KUKA KRL program: GlobalPosn.sub, GlobalPosn.dat

--- GlobalPosn.sub ---
&ACCESS RVO1
&REL 1
&PARAM EDITMASK = *
&PARAM TEMPLATE = C:\KRC\Roboter\Template\submit
DEF  GlobalPosn ( )
; **************************************
; * Package:     TeslaCore             *
; * Release      V4.0.0                *
; * File:        GlobalPosn.sub        *
; * Date:        07.2016               *
; * GUI Version: > = V8.3              *
; **************************************
;FOLD Details
;FOLD Declaration
DECL BOOL bPosEvalResult
;ENDFOLD (Declaration)
LOOP
;FOLD Implementation
;FOLD Position GP1
IF (xGP_Ctrl[1].PosnEnabled==TRUE) THEN
	bPosEvalResult = CheckAxisPos(XGlobal1,xGP_Ctrl[1])
	SetPosOut(bPosEvalResult,xGP_Ctrl[1])
ELSE
   SetPosOut(FALSE,xGP_Ctrl[1])
ENDIF
;ENDFOLD (Position GP1)
;FOLD Position GP2
IF (xGP_Ctrl[2].PosnEnabled==TRUE) THEN
	bPosEvalResult = CheckAxisPos(XGlobal2,xGP_Ctrl[2])
	SetPosOut(bPosEvalResult,xGP_Ctrl[2])
ELSE
   SetPosOut(FALSE,xGP_Ctrl[2])
ENDIF
;ENDFOLD (Position GP2)
;FOLD Position GP3
IF (xGP_Ctrl[3].PosnEnabled==TRUE) THEN
	bPosEvalResult = CheckAxisPos(XGlobal3,xGP_Ctrl[3])
	SetPosOut(bPosEvalResult,xGP_Ctrl[3])
ELSE
   SetPosOut(FALSE,xGP_Ctrl[3])
ENDIF
;ENDFOLD (Position GP3)
;FOLD Position GP4
IF (xGP_Ctrl[4].PosnEnabled==TRUE) THEN
	bPosEvalResult = CheckAxisPos(XGlobal4,xGP_Ctrl[4])
	SetPosOut(bPosEvalResult,xGP_Ctrl[4])
ELSE
   SetPosOut(FALSE,xGP_Ctrl[4])
ENDIF
;ENDFOLD (Position GP4)
;FOLD Position GP5
IF (xGP_Ctrl[5].PosnEnabled==TRUE) THEN
	bPosEvalResult = CheckAxisPos(XGlobal5,xGP_Ctrl[5])
	SetPosOut(bPosEvalResult,xGP_Ctrl[5])
ELSE
   SetPosOut(FALSE,xGP_Ctrl[5])
ENDIF
;ENDFOLD (Position GP5)
;FOLD Position GP6
IF (xGP_Ctrl[6].PosnEnabled==TRUE) THEN
	bPosEvalResult = CheckAxisPos(XGlobal6,xGP_Ctrl[6])
	SetPosOut(bPosEvalResult,xGP_Ctrl[6])
ELSE
   SetPosOut(FALSE,xGP_Ctrl[6])
ENDIF
;ENDFOLD (Position GP6)
;FOLD Position GP7
IF (xGP_Ctrl[7].PosnEnabled==TRUE) THEN
	bPosEvalResult = CheckAxisPos(XGlobal7,xGP_Ctrl[7])
	SetPosOut(bPosEvalResult,xGP_Ctrl[7])
ELSE
   SetPosOut(FALSE,xGP_Ctrl[7])
ENDIF
;ENDFOLD (Position GP7)
;FOLD Position GP8
IF (xGP_Ctrl[8].PosnEnabled==TRUE) THEN
	bPosEvalResult = CheckAxisPos(XGlobal8,xGP_Ctrl[8])
	SetPosOut(bPosEvalResult,xGP_Ctrl[8])
ELSE
   SetPosOut(FALSE,xGP_Ctrl[8])
ENDIF
;ENDFOLD (Position GP8)
;FOLD Position GP9
IF (xGP_Ctrl[9].PosnEnabled==TRUE) THEN
	bPosEvalResult = CheckAxisPos(XGlobal9,xGP_Ctrl[9])
	SetPosOut(bPosEvalResult,xGP_Ctrl[9])
ELSE
   SetPosOut(FALSE,xGP_Ctrl[9])
ENDIF
;ENDFOLD (Position GP9)
;FOLD Position GP10
IF (xGP_Ctrl[10].PosnEnabled==TRUE) THEN
	bPosEvalResult = CheckAxisPos(XGlobal10,xGP_Ctrl[10])
	SetPosOut(bPosEvalResult,xGP_Ctrl[10])
ELSE
   SetPosOut(FALSE,xGP_Ctrl[10])
ENDIF
;ENDFOLD (Position GP10)
;ENDFOLD (Implementation)
ENDLOOP
;ENDFOLD (Details)
END ; (GlobalPosn)

DEFFCT BOOL CheckAxisPos (pPosition: IN, pPosCtrl: IN )
;FOLD Details
;FOLD Declaration
E6Axis pPosition
DECL PosnCtrl_Typ pPosCtrl
BOOL bResult
REAL Angle1, Angle2, Angle3, Angle4, Angle5, Angle6, Angle7, Angle8, Angle9, Angle10, Angle11, Angle12
;ENDFOLD (Declaration)
;FOLD Implementation
IF ((VARSTATE("pPosition") == #INITIALIZED) AND (VARSTATE("pPosCtrl") == #INITIALIZED))THEN
	Angle1 =  ABS(pPosition.A1 - $AXIS_ACT.A1)
	IF (Angle1>pPosCtrl.A1_Tol) THEN
		RETURN(FALSE)
	ENDIF
	Angle2 =  ABS(pPosition.A2 - $AXIS_ACT.A2)
	IF (Angle2>pPosCtrl.A2_Tol) THEN
		RETURN(FALSE)
	ENDIF
	Angle3 =  ABS(pPosition.A3 - $AXIS_ACT.A3)
	IF (Angle3>pPosCtrl.A3_Tol) THEN
		RETURN(FALSE)
	ENDIF
	Angle4 =  ABS(pPosition.A4 - $AXIS_ACT.A4)
	IF (Angle4>pPosCtrl.A4_Tol) THEN
		RETURN(FALSE)
	ENDIF
	Angle5 =  ABS(pPosition.A5 - $AXIS_ACT.A5)
	IF (Angle5>pPosCtrl.A5_Tol) THEN
		RETURN(FALSE)
	ENDIF
	Angle6 =  ABS(pPosition.A6 - $AXIS_ACT.A6)
	IF (Angle6>pPosCtrl.A6_Tol) THEN
		RETURN(FALSE)
	ENDIF
	Angle7 =  ABS(pPosition.E1 - $AXIS_ACT.E1)
	IF (Angle7>pPosCtrl.E1_Tol) THEN
		RETURN(FALSE)
	ENDIF
	Angle8 =  ABS(pPosition.E2 - $AXIS_ACT.E2)
	IF (Angle8>pPosCtrl.E2_Tol) THEN
		RETURN(FALSE)
	ENDIF
	Angle9 =  ABS(pPosition.E3 - $AXIS_ACT.E3)
	IF (Angle9>pPosCtrl.E3_Tol) THEN
		RETURN(FALSE)
	ENDIF
	Angle10 =  ABS(pPosition.E4 - $AXIS_ACT.E4)
	IF (Angle10>pPosCtrl.E4_Tol) THEN
		RETURN(FALSE)
	ENDIF
	Angle11 =  ABS(pPosition.E5 - $AXIS_ACT.E5)
	IF (Angle11>pPosCtrl.E5_Tol) THEN
		RETURN(FALSE)
	ENDIF
	Angle12 =  ABS(pPosition.E6 - $AXIS_ACT.E6)
	IF (Angle12>pPosCtrl.E6_Tol) THEN
		RETURN(FALSE)
	ENDIF
	RETURN (TRUE)
ELSE
	RETURN (FALSE)
ENDIF
;ENDFOLD (Implementation)
;ENDFOLD (Details)
ENDFCT ; (CheckAxisPos)

DEF SetPosOut(bState :IN, pPosCtrl :IN)
;FOLD Details
;FOLD Declaration
BOOL bState
DECL PosnCtrl_Typ pPosCtrl
;ENDFOLD (Declaration)
;FOLD Implementation
IF ((VARSTATE("bState") == #INITIALIZED) AND (VARSTATE("pPosCtrl") == #INITIALIZED))THEN
	IF (pPosCtrl.OutputCtrl > 0) THEN
		IF (pPosCtrl.AtPosn == TRUE) THEN
			$OUT[pPosCtrl.OutputCtrl]=bState
		ELSE
			$OUT[pPosCtrl.OutputCtrl]=NOT(bState)
		ENDIF
	ENDIF
ENDIF
;ENDFOLD (Implementation)
;ENDFOLD (Details)
END ; (SetPosOut)

--- GlobalPosn.dat ---
&ACCESS RVO1
&REL 1
&PARAM EDITMASK = *
&PARAM TEMPLATE = C:\KRC\Roboter\Template\submit
DEFDAT GlobalPosn PUBLIC
; **************************************
; * Package:     TeslaCore             *
; * Release      V4.0.0                *
; * File:        GlobalPosn.dat        *
; * Date:        07.2016               *
; * GUI Version: > = V8.3              *
; **************************************

;FOLD Control Information
DECL GLOBAL INT nMaxGlobalPosn=10 ; Maximum # of global positions
GLOBAL STRUC PosnCtrl_Typ CHAR Comment[24], BOOL PosnEnabled,AtPosn, INT OutputCtrl, REAL A1_Tol, A2_Tol, A3_Tol, A4_Tol, A5_Tol, A6_Tol, E1_Tol, E2_Tol, E3_Tol, E4_Tol, E5_Tol, E6_Tol
DECL GLOBAL PosnCtrl_Typ xGP_Ctrl[10]
xGP_Ctrl[1]={Comment[]" ", PosnEnabled FALSE, AtPosn FALSE, OutputCtrl 0, A1_Tol 2.0, A2_Tol 2.0, A3_Tol 2.0, A4_Tol 2.0, A5_Tol 2.0, A6_Tol 2.0, E1_Tol 2.0, E2_Tol 2.0, E3_Tol 2.0, E4_Tol 2.0, E5_Tol 2.0, E6_Tol 2.0}
xGP_Ctrl[2]={Comment[]" ", PosnEnabled FALSE, AtPosn FALSE,OutputCtrl 0, A1_Tol 2.0, A2_Tol 2.0, A3_Tol 2.0, A4_Tol 2.0, A5_Tol 2.0, A6_Tol 2.0, E1_Tol 2.0, E2_Tol 2.0, E3_Tol 2.0, E4_Tol 2.0, E5_Tol 2.0, E6_Tol 2.0}
xGP_Ctrl[3]={Comment[]" ", PosnEnabled FALSE, AtPosn FALSE,OutputCtrl 0, A1_Tol 2.0, A2_Tol 2.0, A3_Tol 2.0, A4_Tol 2.0, A5_Tol 2.0, A6_Tol 2.0, E1_Tol 2.0, E2_Tol 2.0, E3_Tol 2.0, E4_Tol 2.0, E5_Tol 2.0, E6_Tol 2.0}
xGP_Ctrl[4]={Comment[]" ", PosnEnabled FALSE, AtPosn FALSE,OutputCtrl 0, A1_Tol 2.0, A2_Tol 2.0, A3_Tol 2.0, A4_Tol 2.0, A5_Tol 2.0, A6_Tol 2.0, E1_Tol 2.0, E2_Tol 2.0, E3_Tol 2.0, E4_Tol 2.0, E5_Tol 2.0, E6_Tol 2.0}
xGP_Ctrl[5]={Comment[]" ", PosnEnabled FALSE, AtPosn FALSE,OutputCtrl 0, A1_Tol 2.0, A2_Tol 2.0, A3_Tol 2.0, A4_Tol 2.0, A5_Tol 2.0, A6_Tol 2.0, E1_Tol 2.0, E2_Tol 2.0, E3_Tol 2.0, E4_Tol 2.0, E5_Tol 2.0, E6_Tol 2.0}
xGP_Ctrl[6]={Comment[]" ", PosnEnabled FALSE, AtPosn FALSE,OutputCtrl 0, A1_Tol 2.0, A2_Tol 2.0, A3_Tol 2.0, A4_Tol 2.0, A5_Tol 2.0, A6_Tol 2.0, E1_Tol 2.0, E2_Tol 2.0, E3_Tol 2.0, E4_Tol 2.0, E5_Tol 2.0, E6_Tol 2.0}
xGP_Ctrl[7]={Comment[]" ", PosnEnabled FALSE, AtPosn FALSE,OutputCtrl 0, A1_Tol 2.0, A2_Tol 2.0, A3_Tol 2.0, A4_Tol 2.0, A5_Tol 2.0, A6_Tol 2.0, E1_Tol 2.0, E2_Tol 2.0, E3_Tol 2.0, E4_Tol 2.0, E5_Tol 2.0, E6_Tol 2.0}
xGP_Ctrl[8]={Comment[]" ", PosnEnabled FALSE, AtPosn FALSE,OutputCtrl 0, A1_Tol 2.0, A2_Tol 2.0, A3_Tol 2.0, A4_Tol 2.0, A5_Tol 2.0, A6_Tol 2.0, E1_Tol 2.0, E2_Tol 2.0, E3_Tol 2.0, E4_Tol 2.0, E5_Tol 2.0, E6_Tol 2.0}
xGP_Ctrl[9]={Comment[]" ", PosnEnabled FALSE, AtPosn FALSE,OutputCtrl 0, A1_Tol 2.0, A2_Tol 2.0, A3_Tol 2.0, A4_Tol 2.0, A5_Tol 2.0, A6_Tol 2.0, E1_Tol 2.0, E2_Tol 2.0, E3_Tol 2.0, E4_Tol 2.0, E5_Tol 2.0, E6_Tol 2.0}
xGP_Ctrl[10]={Comment[]" ", PosnEnabled FALSE, AtPosn FALSE,OutputCtrl 0, A1_Tol 2.0, A2_Tol 2.0, A3_Tol 2.0, A4_Tol 2.0, A5_Tol 2.0, A6_Tol 2.0, E1_Tol 2.0, E2_Tol 2.0, E3_Tol 2.0, E4_Tol 2.0, E5_Tol 2.0, E6_Tol 2.0}
;ENDFOLD (Control Information)
;FOLD Positional Information
DECL GLOBAL E6AXIS XGlobal1={A1 0.0,A2 -90.0,A3 90.0,A4 0.0,A5 0.0,A6 0.0,E1 0.0,E2 0.0,E3 0.0,E4 0.0,E5 0.0,E6 0.0}
DECL GLOBAL FDAT FGlobal1={TOOL_NO 1,BASE_NO 0,IPO_FRAME #BASE,POINT2[] " ",TQ_STATE FALSE}
DECL GLOBAL PDAT PGlobal1={VEL 100.000,ACC 100.000,APO_DIST 100.000,GEAR_JERK 50.0000}
DECL GLOBAL LDAT LCGlobal1={VEL 2.00000,ACC 100.000,APO_DIST 100.000,APO_FAC 50.0000,AXIS_VEL 100.000,AXIS_ACC 100.000,ORI_TYP #VAR,CIRC_TYP #BASE,JERK_FAC 50.0000,GEAR_JERK 50.0000,EXAX_IGN 0}

DECL GLOBAL E6AXIS XGlobal2={A1 0.0,A2 -90.0,A3 90.0,A4 0.0,A5 0.0,A6 0.0,E1 0.0,E2 0.0,E3 0.0,E4 0.0,E5 0.0,E6 0.0}
DECL GLOBAL FDAT FGlobal2={TOOL_NO 1,BASE_NO 0,IPO_FRAME #BASE,POINT2[] " ",TQ_STATE FALSE}
DECL GLOBAL PDAT PGlobal2={VEL 100.000,ACC 100.000,APO_DIST 100.000,GEAR_JERK 50.0000}
DECL GLOBAL LDAT LCGlobal2={VEL 2.00000,ACC 100.000,APO_DIST 100.000,APO_FAC 50.0000,AXIS_VEL 100.000,AXIS_ACC 100.000,ORI_TYP #VAR,CIRC_TYP #BASE,JERK_FAC 50.0000,GEAR_JERK 50.0000,EXAX_IGN 0}

DECL GLOBAL E6AXIS XGlobal3={A1 0.0,A2 -90.0,A3 90.0,A4 0.0,A5 0.0,A6 0.0,E1 0.0,E2 0.0,E3 0.0,E4 0.0,E5 0.0,E6 0.0}
DECL GLOBAL FDAT FGlobal3={TOOL_NO 1,BASE_NO 0,IPO_FRAME #BASE,POINT2[] " ",TQ_STATE FALSE}
DECL GLOBAL PDAT PGlobal3={VEL 100.000,ACC 100.000,APO_DIST 100.000,GEAR_JERK 50.0000}
DECL GLOBAL LDAT LCGlobal3={VEL 2.00000,ACC 100.000,APO_DIST 100.000,APO_FAC 50.0000,AXIS_VEL 100.000,AXIS_ACC 100.000,ORI_TYP #VAR,CIRC_TYP #BASE,JERK_FAC 50.0000,GEAR_JERK 50.0000,EXAX_IGN 0}

DECL GLOBAL E6AXIS XGlobal4={A1 0.0,A2 -90.0,A3 90.0,A4 0.0,A5 0.0,A6 0.0,E1 0.0,E2 0.0,E3 0.0,E4 0.0,E5 0.0,E6 0.0}
DECL GLOBAL FDAT FGlobal4={TOOL_NO 1,BASE_NO 0,IPO_FRAME #BASE,POINT2[] " ",TQ_STATE FALSE}
DECL GLOBAL PDAT PGlobal4={VEL 100.000,ACC 100.000,APO_DIST 100.000,GEAR_JERK 50.0000}
DECL GLOBAL LDAT LCGlobal4={VEL 2.00000,ACC 100.000,APO_DIST 100.000,APO_FAC 50.0000,AXIS_VEL 100.000,AXIS_ACC 100.000,ORI_TYP #VAR,CIRC_TYP #BASE,JERK_FAC 50.0000,GEAR_JERK 50.0000,EXAX_IGN 0}

DECL GLOBAL E6AXIS XGlobal5={A1 0.0,A2 -90.0,A3 90.0,A4 0.0,A5 0.0,A6 0.0,E1 0.0,E2 0.0,E3 0.0,E4 0.0,E5 0.0,E6 0.0}
DECL GLOBAL FDAT FGlobal5={TOOL_NO 1,BASE_NO 0,IPO_FRAME #BASE,POINT2[] " ",TQ_STATE FALSE}
DECL GLOBAL PDAT PGlobal5={VEL 100.000,ACC 100.000,APO_DIST 100.000,GEAR_JERK 50.0000}
DECL GLOBAL LDAT LCGlobal5={VEL 2.00000,ACC 100.000,APO_DIST 100.000,APO_FAC 50.0000,AXIS_VEL 100.000,AXIS_ACC 100.000,ORI_TYP #VAR,CIRC_TYP #BASE,JERK_FAC 50.0000,GEAR_JERK 50.0000,EXAX_IGN 0}

DECL GLOBAL E6AXIS XGlobal6={A1 0.0,A2 -90.0,A3 90.0,A4 0.0,A5 0.0,A6 0.0,E1 0.0,E2 0.0,E3 0.0,E4 0.0,E5 0.0,E6 0.0}
DECL GLOBAL FDAT FGlobal6={TOOL_NO 1,BASE_NO 0,IPO_FRAME #BASE,POINT2[] " ",TQ_STATE FALSE}
DECL GLOBAL PDAT PGlobal6={VEL 100.000,ACC 100.000,APO_DIST 100.000,GEAR_JERK 50.0000}
DECL GLOBAL LDAT LCGlobal6={VEL 2.00000,ACC 100.000,APO_DIST 100.000,APO_FAC 50.0000,AXIS_VEL 100.000,AXIS_ACC 100.000,ORI_TYP #VAR,CIRC_TYP #BASE,JERK_FAC 50.0000,GEAR_JERK 50.0000,EXAX_IGN 0}

DECL GLOBAL E6AXIS XGlobal7={A1 0.0,A2 -90.0,A3 90.0,A4 0.0,A5 0.0,A6 0.0,E1 0.0,E2 0.0,E3 0.0,E4 0.0,E5 0.0,E6 0.0}
DECL GLOBAL FDAT FGlobal7={TOOL_NO 1,BASE_NO 0,IPO_FRAME #BASE,POINT2[] " ",TQ_STATE FALSE}
DECL GLOBAL PDAT PGlobal7={VEL 100.000,ACC 100.000,APO_DIST 100.000,GEAR_JERK 50.0000}
DECL GLOBAL LDAT LCGlobal7={VEL 2.00000,ACC 100.000,APO_DIST 100.000,APO_FAC 50.0000,AXIS_VEL 100.000,AXIS_ACC 100.000,ORI_TYP #VAR,CIRC_TYP #BASE,JERK_FAC 50.0000,GEAR_JERK 50.0000,EXAX_IGN 0}

DECL GLOBAL E6AXIS XGlobal8={A1 0.0,A2 -90.0,A3 90.0,A4 0.0,A5 0.0,A6 0.0,E1 0.0,E2 0.0,E3 0.0,E4 0.0,E5 0.0,E6 0.0}
DECL GLOBAL FDAT FGlobal8={TOOL_NO 1,BASE_NO 0,IPO_FRAME #BASE,POINT2[] " ",TQ_STATE FALSE}
DECL GLOBAL PDAT PGlobal8={VEL 100.000,ACC 100.000,APO_DIST 100.000,GEAR_JERK 50.0000}
DECL GLOBAL LDAT LCGlobal8={VEL 2.00000,ACC 100.000,APO_DIST 100.000,APO_FAC 50.0000,AXIS_VEL 100.000,AXIS_ACC 100.000,ORI_TYP #VAR,CIRC_TYP #BASE,JERK_FAC 50.0000,GEAR_JERK 50.0000,EXAX_IGN 0}

DECL GLOBAL E6AXIS XGlobal9={A1 0.0,A2 -90.0,A3 90.0,A4 0.0,A5 0.0,A6 0.0,E1 0.0,E2 0.0,E3 0.0,E4 0.0,E5 0.0,E6 0.0}
DECL GLOBAL FDAT FGlobal9={TOOL_NO 1,BASE_NO 0,IPO_FRAME #BASE,POINT2[] " ",TQ_STATE FALSE}
DECL GLOBAL PDAT PGlobal9={VEL 100.000,ACC 100.000,APO_DIST 100.000,GEAR_JERK 50.0000}
DECL GLOBAL LDAT LCGlobal9={VEL 2.00000,ACC 100.000,APO_DIST 100.000,APO_FAC 50.0000,AXIS_VEL 100.000,AXIS_ACC 100.000,ORI_TYP #VAR,CIRC_TYP #BASE,JERK_FAC 50.0000,GEAR_JERK 50.0000,EXAX_IGN 0}

DECL GLOBAL E6AXIS XGlobal10={A1 0.0,A2 -90.0,A3 90.0,A4 0.0,A5 0.0,A6 0.0,E1 0.0,E2 0.0,E3 0.0,E4 0.0,E5 0.0,E6 0.0}
DECL GLOBAL FDAT FGlobal10={TOOL_NO 1,BASE_NO 0,IPO_FRAME #BASE,POINT2[] " ",TQ_STATE FALSE}
DECL GLOBAL PDAT PGlobal10={VEL 100.000,ACC 100.000,APO_DIST 100.000,GEAR_JERK 50.0000}
DECL GLOBAL LDAT LCGlobal10={VEL 2.00000,ACC 100.000,APO_DIST 100.000,APO_FAC 50.0000,AXIS_VEL 100.000,AXIS_ACC 100.000,ORI_TYP #VAR,CIRC_TYP #BASE,JERK_FAC 50.0000,GEAR_JERK 50.0000,EXAX_IGN 0}
;ENDFOLD (Positional Information)

ENDDAT
